Fanuc KAREL source: kb00024.compact.KL

PROGRAM KB00024
%STACKSIZE=65535
%PRIORITY=65535
%NOLOCKGROUP
VAR
P1 : FILE
BEGIN
CLR_IO_STAT(P1)
END KB00024
